FUNCTION_BLOCK INTERFACE_HTTP (* Peroidic event generator *)
  (* Standard: 61499-1 Annex A; Description: Copyright (c) 2017 fortiss GmbH This program and the accompanying materials are made available under the terms of the Eclipse Public License 2.0 which is available at https://www.eclipse.org/legal/epl-2.0/ SPDX-License-Identifier: EPL-2.0 *)
  (* Version 1.0, 2017-09-21, Alois Zoitl, fortiss GmbH, initial API and implementation and/or initial documentation *)
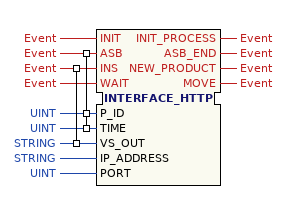
  EVENT_INPUT
    INIT;
    ASB WITH P_ID, TIME;
    INS WITH VS_OUT;
    WAIT;
  END_EVENT
  EVENT_OUTPUT
    INIT_PROCESS;
    ASB_END;
    NEW_PRODUCT;
    MOVE;
  END_EVENT
  VAR_INPUT
    P_ID : UINT;
    TIME : UINT;
    VS_OUT : STRING;
    IP_ADDRESS : STRING;
    PORT : UINT;
  END_VAR
END_FUNCTION_BLOCK
